Fanuc KAREL source: kb00081.KL

PROGRAM KB00081
%STACKSIZE=65535
%PRIORITY=65535
%NOLOCKGROUP
VAR
P1 : INTEGER
P2 : INTEGER
P3 : INTEGER
RESULT : INTEGER
BEGIN
P1=1
P2=1
P3=1
RESULT=GET_PORT_ATR(P1,P2,P3)
END KB00081
